// TIA Portal V21 export
// export: Created 2026-07-28T16:54:16.2898592Z, ExportSetting WithDefaults, DisplayName Totally Integrated Automation Portal, DisplayVersion V21, DisplayName SINAMICS Startdrive Advanced, DisplayVersion V21, DisplayName SINAMICS Startdrive G110M, G120, G120C, G120D, G120P, G115D, DisplayVersion V21, DisplayName SINAMICS Startdrive G130, G150, S120, S150, G200, G220, S200, S210, S220, Innomotics MVD, DisplayVersion V21, DisplayName STEP 7 Professional, DisplayVersion V21, DisplayName STEP 7 Safety, DisplayVersion V21, DisplayName Tech WebApplication, DisplayVersion V21, DisplayName WinCC Basic/Comfort/Advanced, DisplayVersion V21, DisplayName WinCC Professional, DisplayVersion V21, DisplayName WinCC Unified, DisplayVersion V21
DATA_BLOCK "DB GLOBAL"   // DB1
{ S7_Optimized_Access := 'TRUE' }
VERSION : 0.1
// Esqueleto -- so a forma que os geradores exigem, nenhum dado de projeto.
//  Importar DEPOIS de MotorDados/ValvDados (referencia os dois).
// 
//  Contrato consumido pelos geradores:
//    gen-alarm-fc  -> "DB GLOBAL".<AREA>.ALARMES.WORD_ALARMES_<n>, n a partir de 1
//                     (AlarmFc.cs:282; a area e achada por nome em AlarmFc.FindParentStruct)
//    gen-fault-ob  -> "DB GLOBAL".HARDWARE_INTERRUPT.ALARMES_MODULOS.<QA-xx>.WORD_<n>.%X<bit>
//                     (FaultOb.cs:23, uma word por 16 modulos do rack)
//  Uma area por secao da planta; duplicar o bloco AREA_01 e renomear.
// stored: AutoNumber true, IsOnlyStoredInLoadMemory false, IsWriteProtectedInAS false
   VAR
      AREA_01 : Struct
         ALARMES : Struct
            WORD_ALARMES_1 : Word;
            WORD_ALARMES_2 : Word;
            WORD_ALARMES_3 : Word;
            WORD_ALARMES_4 : Word;
            WORD_ALARMES_5 : Word;
            WORD_ALARMES_6 : Word;
            WORD_ALARMES_7 : Word;
            WORD_ALARMES_8 : Word;   // equipamentos da area -- o gerador de FC de alarme casa o nome do tag com o nome do membro pra descobrir a que area o alarme pertence
         END_STRUCT;
         BOMBA_01 { S7_SetPoint := 'True'} : "MotorDados";
         VALVULA_01 { S7_SetPoint := 'True'} : "ValvDados";
      END_STRUCT;
      HARDWARE_INTERRUPT : Struct
         ALARMES_MODULOS : Struct
            "QA-00" : Struct   // um struct por painel/rack de I/O
               WORD_1 : Word;
               WORD_2 : Word;
            END_STRUCT;
            "QA-01" : Struct
               WORD_1 : Word;
               WORD_2 : Word;
            END_STRUCT;
         END_STRUCT;
      END_STRUCT;
   END_VAR
BEGIN
END_DATA_BLOCK
